// TIA Portal project "4_Pick_n_Place" (V19)

(* hardware
DEVICE "S7-1500/ET200MP station_1"  S7-1500 station
   slot 0: "Rail_0"  Rack  6ES7 590-1***0-0AA0
   slot 1: "PLC_1"  CPU 1513-1 PN  6ES7 513-1AL02-0AB0  V2.9
      slot 3: "CPU display_1"  6ES7591-1AA00-0AA0
      slot 32768: "PROFINET interface_1"  X1
         slot 32769: "Port_1"  X1 P1
         slot 32770: "Port_2"  X1 P2
      slot 34817: "Virtual CP interface port_1"  Virtual CP interface port  Virtual CP interface port
*)

// ===== PLC "PLC_1"  CPU 1513-1 PN =====

VAR_GLOBAL   // PLC tag table "Default tag table"
   "Step" AT %MD0 : DInt;
   "Tag_1" AT %M0.0 : Bool;
   "Buffer_Item at exit" AT %M0.1 : Bool;
   "Tag_2" AT %M0.2 : Bool;
END_VAR

VAR_GLOBAL   // PLC tag table "Tag table from XML_1"
   "Start" AT %I0.0 : Bool;
   "Stop" AT %I0.1 : Bool;
   "Item at entry" AT %I0.2 : Bool;
   "Item at exit" AT %I0.3 : Bool;
   "Moving X" AT %I0.4 : Bool;
   "Moving Z" AT %I0.5 : Bool;
   "Item detected" AT %I0.6 : Bool;
   "Start light" AT %Q0.0 : Bool;
   "Stop light" AT %Q0.1 : Bool;
   "Entry conveyor" AT %Q0.2 : Bool;
   "Exit conveyor" AT %Q0.3 : Bool;
   "Move X" AT %Q0.4 : Bool;
   "Move Z" AT %Q0.5 : Bool;
   "Grab" AT %Q0.6 : Bool;
   "Counter" AT %QD30 : DInt;
END_VAR

// folder: System blocks/Program resources

DATA_BLOCK "IEC_Timer_0_DB"   // DB1
{ S7_Optimized_Access := 'TRUE' }
AUTHOR : Simatic
FAMILY : IEC
NAME : IEC_TMR
VERSION : 1.0
// stored: InstanceOfName IEC_TIMER
"IEC_TIMER"
BEGIN
END_DATA_BLOCK

DATA_BLOCK "IEC_Counter_0_DB"   // DB2
{ S7_Optimized_Access := 'TRUE' }
AUTHOR : Simatic
FAMILY : IEC
NAME : CNTR
VERSION : 1.0
// stored: InstanceOfName IEC_COUNTER
"IEC_COUNTER"
BEGIN
END_DATA_BLOCK

DATA_BLOCK "IEC_Timer_0_DB_1"   // DB3
{ S7_Optimized_Access := 'TRUE' }
AUTHOR : Simatic
FAMILY : IEC
NAME : IEC_TMR
VERSION : 1.0
// stored: InstanceOfName IEC_TIMER
"IEC_TIMER"
BEGIN
END_DATA_BLOCK

DATA_BLOCK "IEC_Timer_0_DB_2"   // DB4
{ S7_Optimized_Access := 'TRUE' }
AUTHOR : Simatic
FAMILY : IEC
NAME : IEC_TMR
VERSION : 1.0
// stored: InstanceOfName IEC_TIMER
"IEC_TIMER"
BEGIN
END_DATA_BLOCK

// folder: (top level)

ORGANIZATION_BLOCK "Main"   // OB1, LAD, ProgramCycle
TITLE = "Main Program Sweep (Cycle)"
{ S7_Optimized_Access := 'TRUE' }
VERSION : 0.1
   VAR_INPUT
      Initial_Call : Bool;   // Initial call of this OB
      Remanence : Bool;   // =True, if remanent data are available
   END_VAR
   VAR_TEMP   // added for the SCL form of the ladder/FBD networks
      _w1 : Bool;
   END_VAR
BEGIN

REGION Network 1: Start the light, if item not in entry and not grab, run the entry conveyor, if item at entry, and not grab, move the z axis down
   // Start the light, if item not in entry and not grab, run the entry conveyor, if item at entry, and not grab, move the z axis down
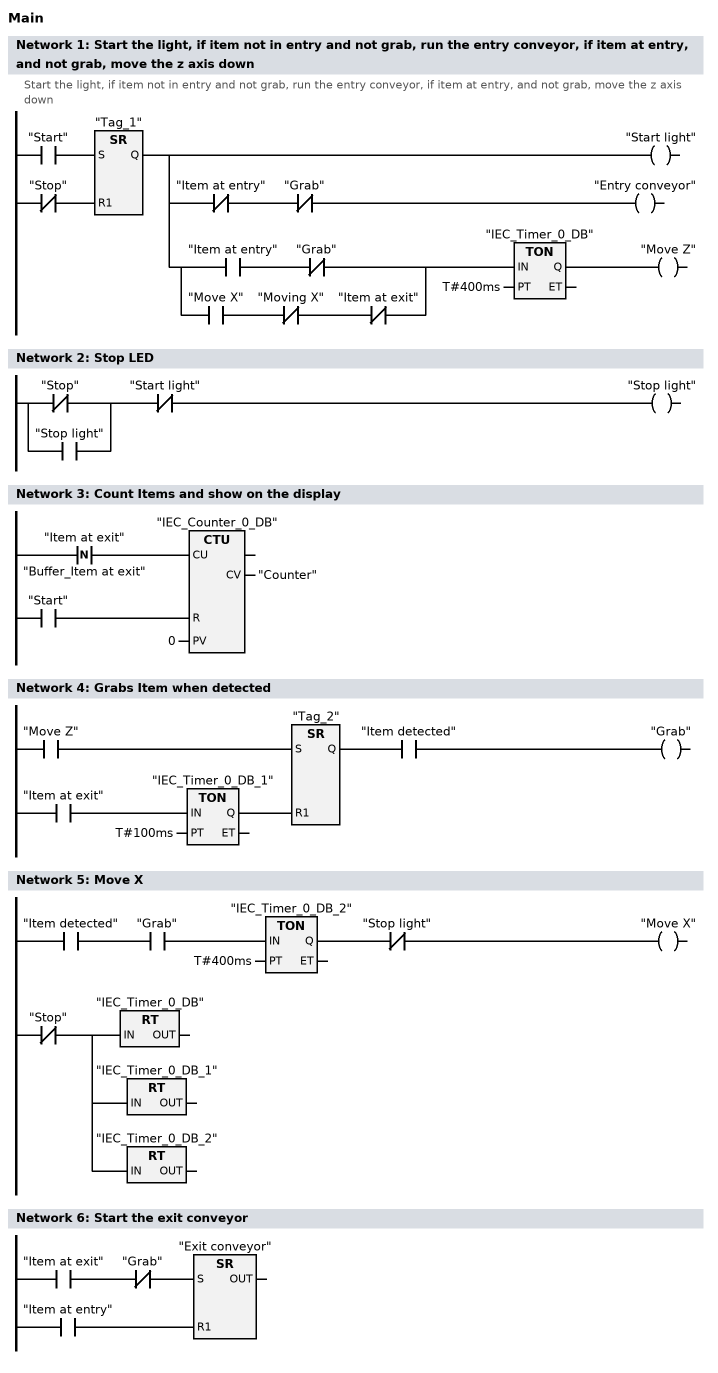
   IF "Start" THEN
       "Tag_1" := TRUE;   // SR flip-flop
   END_IF;
   IF NOT "Stop" THEN "Tag_1" := FALSE; END_IF;
   "Start light" := "Tag_1";
   "Entry conveyor" := "Tag_1" AND NOT "Item at entry" AND NOT "Grab";
   "IEC_Timer_0_DB".TON(IN := "Tag_1" AND (("Item at entry" AND NOT "Grab") OR ("Move X" AND NOT "Moving X" AND NOT "Item at exit")),
                        PT := T#400ms);
   "Move Z" := "IEC_Timer_0_DB".Q;
END_REGION

REGION Network 2: Stop LED
   RUNG wire#powerrail
      I_Contact( "Stop" )
      wire#w1
      I_Contact( "Start light" )
      Coil( "Stop light" )
   END_RUNG
   RUNG wire#powerrail
      Contact( "Stop light" )
   END_RUNG wire#w1
   // the same network as SCL:
   "Stop light" := (NOT "Stop" OR "Stop light") AND NOT "Start light";
END_REGION

REGION Network 3: Count Items and show on the display
   #_w1 := NOT "Item at exit" AND "Buffer_Item at exit";   // falling edge of "Item at exit"
   "Buffer_Item at exit" := "Item at exit";
   "IEC_Counter_0_DB".CTU(CU := #_w1, R := "Start", PV := 0, CV => "Counter");
END_REGION

REGION Network 4: Grabs Item when detected
   "IEC_Timer_0_DB_1".TON(IN := "Item at exit", PT := T#100ms);
   IF "Move Z" THEN
       "Tag_2" := TRUE;   // SR flip-flop
   END_IF;
   IF "IEC_Timer_0_DB_1".Q THEN "Tag_2" := FALSE; END_IF;
   "Grab" := "Tag_2" AND "Item detected";
END_REGION

REGION Network 5: Move X
   "IEC_Timer_0_DB_2".TON(IN := "Item detected" AND "Grab", PT := T#400ms);
   "Move X" := "IEC_Timer_0_DB_2".Q AND NOT "Stop light";
   IF NOT "Stop" THEN
       RESET_TIMER("IEC_Timer_0_DB");
       RESET_TIMER("IEC_Timer_0_DB_1");
       RESET_TIMER("IEC_Timer_0_DB_2");
   END_IF;
END_REGION

REGION Network 6: Start the exit conveyor
   RUNG wire#powerrail
      Contact( "Item at exit" )
      I_Contact( "Grab" )
      S_SR(operand := "Exit conveyor", r1 := wire#w1)
   END_RUNG
   RUNG wire#powerrail
      Contact( "Item at entry" )
   END_RUNG wire#w1
   // the same network as SCL:
   IF "Item at exit" AND NOT "Grab" THEN
       "Exit conveyor" := TRUE;   // SR flip-flop
   END_IF;
   IF "Item at entry" THEN "Exit conveyor" := FALSE; END_IF;
END_REGION
END_ORGANIZATION_BLOCK